FUNCTION_BLOCK CountPulse (* Basic Function Block Type *)
  (* Standard: 61499-2 *)
  (* Version 0.0, 8/6/2026, Schneider Electric, Template *)
  PACKAGE SE.Nereda;
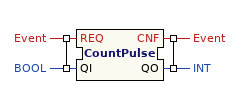
  EVENT_INPUT
    REQ WITH QI; (* Normal Execution Request *)
  END_EVENT
  EVENT_OUTPUT
    CNF WITH QO; (* Execution Confirmation *)
  END_EVENT
  VAR_INPUT
    QI : BOOL; (* Input event qualifier *)
  END_VAR
  VAR_OUTPUT
    QO : INT; (* Output event qualifier *)
  END_VAR
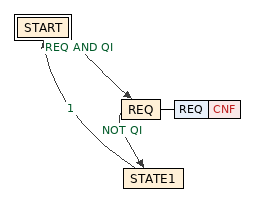
  EC_STATES
    START; (* Initial State *)
    REQ : REQ -> CNF; (* Normal execution *)
    STATE1;
  END_STATES
  EC_TRANSITIONS
    START TO REQ := REQ AND QI;
    STATE1 TO START := 1;
    REQ TO STATE1 := NOT QI;
  END_TRANSITIONS
  ALGORITHM REQ IN ST: (* Normally executed algorithm *)
;
IF QO < 9999 THEN
	QO := QO + 1;
ELSE
	QO := 0;
END_IF;
  END_ALGORITHM
END_FUNCTION_BLOCK
